FUNCTION_BLOCK FC_HeatingCurve_Test EXTENDS FB_TestSuite
VAR

END_VAR

TAmbNegative();
TAmbZero();
HeatingCurveZero();
HeatingCurveNegative();

METHOD HeatingCurveNegative // This method checks whether the heating curve can have a negative value
VAR
	HeatingCurveRes: Real;		//Actual value for Heating Curve
	ExpectedValue : REAL := -1;	//Expected value for Heating Curve
	fSlope: REAL := -1;				//Slope of Heating Curve
	fOffset: REAL := 35;				//Offset of Heating Curve

END_VAR
TEST('HeatingCurveNegative');
 
HeatingCurveRes := FC_HeatingCurve(fTempAmb := 36, fSlope, fOffset);
 
AssertEquals(Expected := ExpectedValue,
             Actual := HeatingCurveRes,
             Message := 'The calculation is not correct');
 
TEST_FINISHED();
END_METHOD

METHOD HeatingCurveZero // This method checks whether the heating curve can have zero as value
VAR
	HeatingCurveRes: REAL;		//Actual value for Heating Curve
	ExpectedValue : REAL := 0;  //Expected value for Heating Curve
	fSlope: REAL := -1;				//Slope of Heating Curve
	fOffset: REAL := 35;				//Offset of Heating Curve
//	fTempAmb: REAL

END_VAR
TEST('HeatingCurveZero');
 
HeatingCurveRes := FC_HeatingCurve(fTempAmb := 35, fSlope, fOffset);
 
AssertEquals(Expected := ExpectedValue,
             Actual := HeatingCurveRes,
             Message := 'The calculation is not correct');
 
TEST_FINISHED();
END_METHOD

METHOD TAmbNegative // This method checks whether negative ambient temperatures work properly
VAR
	HeatingCurveRes: REAL;		 //Actual value for Heating Curve
	ExpectedValue : REAL := 40;  //Expected value for Heating Curve
	fSlope: REAL := -1;				 //Slope of Heating Curve
	fOffset: REAL := 35;				 //Offset of Heating Curve
END_VAR
TEST('TAmbNegative');
 
HeatingCurveRes := FC_HeatingCurve(fTempAmb := -5, fSlope, fOffset);
 
AssertEquals(Expected := ExpectedValue,
             Actual := HeatingCurveRes,
             Message := 'The calculation is not correct');
 
TEST_FINISHED();
END_METHOD

METHOD TAmbZero // This method checks whether zero degrees as ambient temperature work properly
VAR
	HeatingCurveRes : REAL;		  //Actual value for Heating Curve
	ExpectedValue : REAL := 35;   //Expected value for Heating Curve
	fSlope: REAL := -1;				  //Slope of Heating Curve	
	fOffset: REAL := 35;				  //Offset of Heating Curve

END_VAR
TEST('TAmbZero');
 
HeatingCurveRes := FC_HeatingCurve(fTempAmb := 0, fSlope, fOffset);
 
AssertEquals(Expected := ExpectedValue,
             Actual := HeatingCurveRes,
             Message := 'The calculation is not correct');
 
TEST_FINISHED();
END_METHOD

END_FUNCTION_BLOCK

(* stored: Version 1.1.0.1, ProductVersion 3.1.4024.6
   POU FC_HeatingCurve_Test: Id {83922ca9-fec5-4955-81a6-65a3cfbdb7ba}, SpecialFunc None
   Method HeatingCurveNegative: Id {a051f6a0-e43e-4c8d-bd11-4cf8c3ba617f}
   Method HeatingCurveZero: Id {09c65531-87c1-4c8d-979f-ab1b51070c4f}
   Method TAmbNegative: Id {738f967b-eb89-490a-9e92-7f198ccd229a}
   Method TAmbZero: Id {7792e1b4-7c9f-44f8-830b-ec1144c32ab4} *)
